VAR_GLOBAL
    //Better have your inputs and outputs!
    // M1K4
    Serial_stComIn_M1K4   AT %I*	:	EL6inData22B (*KL6inData22B*);
    Serial_stComOut_M1K4  AT %Q*	:	EL6outData22B (*KL6outData22B*);
END_VAR

(* stored: Version 1.1.0.1, ProductVersion 3.1.4022.18
   GVL GVL_SerialIO: Id {c473b3fd-251c-4dab-9486-f893066a90f0} *)
